{attribute 'linkalways'} 
{attribute 'no_explicit_call' := 'This FB is a CLASS and must be accessed using methods or properties'}
{attribute 'enable_dynamic_creation'}
FUNCTION_BLOCK GetDatatypesRpcHandler IMPLEMENTS I_RpcHandler
VAR
	datatypes : I_Datatypes;
END_VAR

METHOD Handle
VAR_INPUT
	Parameters : I_Deserializer;
	Response : I_SynchronousRpcResponse;
END_VAR
VAR
	serializer : I_Serializer;
END_VAR
IF datatypes = 0 THEN
	Response.RejectWithMessage('GetDatatypesRpcHandler has not been initialized with a valid datatypes object');
	RETURN;
END_IF

serializer := Response.GetSerializer();
datatypes.SerializeTypeWith(serializer);
Response.CompleteWithSerializer(serializer);
serializer.Dispose();
END_METHOD

METHOD PUBLIC Initialize
VAR_INPUT
	Datatypes : I_Datatypes;
END_VAR
this^.datatypes := Datatypes;
END_METHOD

END_FUNCTION_BLOCK

(* stored: Version 1.1.0.1, ProductVersion 3.1.4024.12
   POU GetDatatypesRpcHandler: Id {e14e6668-de45-4ee4-b72a-10a786028e2f}, SpecialFunc None
   Method Handle: Id {b323c91b-c631-4242-8b5b-8446f49cc41e}
   Method Initialize: Id {b88efccc-de3d-4953-858d-990b9af491f9} *)
